Staubli VAL3: refresh.pgx

program refresh()
// // page refresh
  local string l_sMessage
begin
  if !bShowMessage
    if (nKey>=270 and nKey<=278) or abs(clock()-nRefresh)>nTime
      // refresh the static message
      use:bUseRefresh=true
      call refreshDynamic()
    else
      // refresh the Dynamic message
      if use:bUseRefresh
        call refreshDynamic()
      endIf
    endIf
  endIf
  // show the message
  call showMessage()
  // print the instruction
  call printToShow()
end
